FUNCTION TryConvert_LWORD_TO_ULINT : BOOL
VAR_INPUT
	in : LWORD;
	out : REFERENCE TO ULINT;
END_VAR

out := LWORD_TO_ULINT(in);
TryConvert_LWORD_TO_ULINT := TRUE;

END_FUNCTION

(* stored: Version 1.1.0.1, ProductVersion 3.1.4024.12
   POU TryConvert_LWORD_TO_ULINT: Id {a263e698-5c56-4778-be68-7f34aea492c3}, SpecialFunc None *)
